TYPE U_GC_HW_Out :
UNION
	Terminal AT%Q* : ST_GC_Terminal_Out;
	Signal : ST_GC_Signal_Out;
END_UNION
END_TYPE

(* stored: Version 1.1.0.1, ProductVersion 3.1.4026.18
   DUT U_GC_HW_Out: Id {b02ecd0a-ab03-405e-97cd-6b884f7368f9} *)
